(* CODESYS project Prova_CTU.project

Project tree, tasks and I/O mapping:
  Device : CODESYS Control Win V3, 3S - Smart Software Solutions GmbH, order no. 305021, version 3.5.10.30
    application Application
      libraries: Standard, * (System)
      task MainTask (cyclic, interval t#20ms, priority 1) calls PLC_PRG
      task VISU_TASK (cyclic, interval 100 ms, priority 31) calls VisuElems.Visu_Prg
      program PLC_PRG [FBD]
      visualisation Visualization
  text list GlobalTextList
*)

// Device/Application/PLC_PRG
PROGRAM PLC_PRG
VAR
	CTU_0: CTU;
	Contact1: BOOL;
	Debug_CV: WORD;
	Contact2: BOOL;
	Value1: WORD := 3;
END_VAR

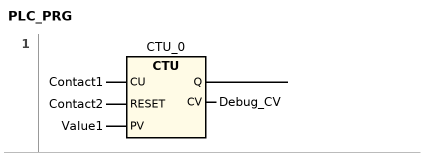
// NETWORK 1
CTU_0(CU := Contact1, RESET := Contact2, PV := Value1, CV => Debug_CV); // CTU

END_PROGRAM

// Device/Application/Visualization
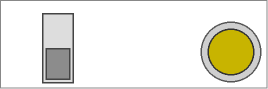
VISUALIZATION Visualization  // 268x89
    Lamp1 (196,17 70x70), variable: PLC_PRG.CTU_0.Q, style: Lamp-Lamp1-Yellow
    DipSwitch (23,13 70x70), variable: PLC_PRG.Contact1, behaviour: TOGGLE, style: Switch-DipSwitch-Gray
END_VISUALIZATION
